// TIA Portal project "PrensaPiezas" (V18)

(* hardware
DEVICE "S7-1200 station_1"  S7-1200 Station
   slot 0: "Rack_0"  S7-1200 Rack  Rack  V1.0
   slot 1: "PLC_1"  CPU 1214C AC/DC/Rly  6ES7 214-1BG40-0XB0  V4.6
*)

// ===== PLC "PLC_1"  CPU 1214C AC/DC/Rly =====

VAR_GLOBAL   // PLC tag table "Default tag table"
   "rampa" AT %I0.0 : Bool;   // Sensor del objeto al caer de la rampa
   "zonaPrensa" AT %I0.1 : Bool;   // Sensor de la zona de la prensa
   "piezaPosicion" AT %I0.2 : Bool;   // Sensor de la pieza en posicion
   "prensa" AT %I0.3 : Bool;   // Sensor de la prensa
   "finalTramo" AT %I0.4 : Bool;   // Sensor del tramo final de la cinta
   "cintaAvanza" AT %M0.0 : Bool;   // Marca para avanzar la cinta
   "centraPieza" AT %M0.1 : Bool;   // Marca para centrar la pieza
   "cilindroBaja" AT %M0.2 : Bool;   // Marca para accionar la prensa
   "cintaRetrocede" AT %M0.3 : Bool;   // Marca para retroceder la cinta
   "guiaFlanco" AT %M0.4 : Bool;   // Marca guia de flanco
   "guiaFlanco_1" AT %M0.5 : Bool;   // Marca guia de flanco
   "guiaFlanco_2" AT %M0.6 : Bool;   // Marca guia de flanco
   "guiaFlanco_3" AT %M0.7 : Bool;   // Marca guia de flanco
   "motor" AT %Q0.0 : Bool;   // Motor hacia delante
   "motor_2" AT %Q0.1 : Bool;   // Motor hacia atras
   "presadoPieza" AT %Q0.2 : Bool;   // Prensado a la pieza
   "centrarPieza" AT %Q0.3 : Bool;   // Centrador de la pieza
END_VAR

// folder: System blocks/Program resources

DATA_BLOCK "retardoPiezaPresado"   // DB1
{ S7_Optimized_Access := 'TRUE' }
AUTHOR : Simatic
FAMILY : IEC
NAME : IEC_TMR
VERSION : 1.0
// stored: InstanceOfName IEC_TIMER
"IEC_TIMER"
BEGIN
END_DATA_BLOCK

// folder: (top level)

ORGANIZATION_BLOCK "Main"   // OB1, LAD, ProgramCycle
TITLE = "Main Program Sweep (Cycle)"
{ S7_Optimized_Access := 'TRUE' }
VERSION : 0.1
   VAR_INPUT
      Initial_Call : Bool;   // Initial call of this OB
      Remanence : Bool;   // =True, if remanent data are available
   END_VAR
   VAR_TEMP   // added for the SCL form of the ladder/FBD networks
      _w1 : Bool;
      _w2 : Bool;
   END_VAR
BEGIN

REGION Network 1: Marca para avanzar la cinta
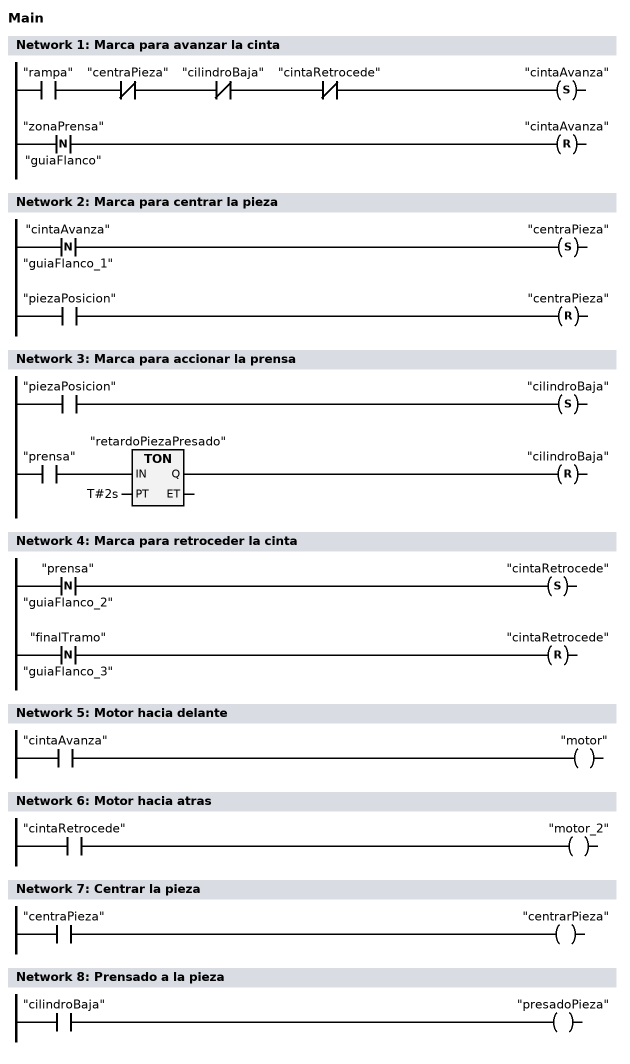
   RUNG wire#powerrail
      Contact( "rampa" )
      I_Contact( "centraPieza" )
      I_Contact( "cilindroBaja" )
      I_Contact( "cintaRetrocede" )
      S_Coil( "cintaAvanza" )
   END_RUNG
   RUNG wire#powerrail
      N_Contact(operand := "zonaPrensa", bit := "guiaFlanco")
      R_Coil( "cintaAvanza" )
   END_RUNG
   // the same network as SCL:
   IF "rampa" AND NOT "centraPieza" AND NOT "cilindroBaja" AND NOT "cintaRetrocede" THEN
       "cintaAvanza" := TRUE;
   END_IF;
   #_w1 := NOT "zonaPrensa" AND "guiaFlanco";   // falling edge of "zonaPrensa"
   "guiaFlanco" := "zonaPrensa";
   IF #_w1 THEN "cintaAvanza" := FALSE; END_IF;
END_REGION

REGION Network 2: Marca para centrar la pieza
   RUNG wire#powerrail
      N_Contact(operand := "cintaAvanza", bit := "guiaFlanco_1")
      S_Coil( "centraPieza" )
   END_RUNG
   RUNG wire#powerrail
      Contact( "piezaPosicion" )
      R_Coil( "centraPieza" )
   END_RUNG
   // the same network as SCL:
   #_w1 := NOT "cintaAvanza" AND "guiaFlanco_1";   // falling edge of "cintaAvanza"
   "guiaFlanco_1" := "cintaAvanza";
   IF #_w1 THEN "centraPieza" := TRUE; END_IF;
   IF "piezaPosicion" THEN "centraPieza" := FALSE; END_IF;
END_REGION

REGION Network 3: Marca para accionar la prensa
   IF "piezaPosicion" THEN "cilindroBaja" := TRUE; END_IF;
   "retardoPiezaPresado".TON(IN := "prensa", PT := T#2s);
   IF "retardoPiezaPresado".Q THEN "cilindroBaja" := FALSE; END_IF;
END_REGION

REGION Network 4: Marca para retroceder la cinta
   RUNG wire#powerrail
      N_Contact(operand := "prensa", bit := "guiaFlanco_2")
      S_Coil( "cintaRetrocede" )
   END_RUNG
   RUNG wire#powerrail
      N_Contact(operand := "finalTramo", bit := "guiaFlanco_3")
      R_Coil( "cintaRetrocede" )
   END_RUNG
   // the same network as SCL:
   #_w1 := NOT "prensa" AND "guiaFlanco_2";   // falling edge of "prensa"
   "guiaFlanco_2" := "prensa";
   IF #_w1 THEN "cintaRetrocede" := TRUE; END_IF;
   #_w2 := NOT "finalTramo" AND "guiaFlanco_3";   // falling edge of "finalTramo"
   "guiaFlanco_3" := "finalTramo";
   IF #_w2 THEN "cintaRetrocede" := FALSE; END_IF;
END_REGION

REGION Network 5: Motor hacia delante
   RUNG wire#powerrail
      Contact( "cintaAvanza" )
      Coil( "motor" )
   END_RUNG
   // the same network as SCL:
   "motor" := "cintaAvanza";
END_REGION

REGION Network 6: Motor hacia atras
   RUNG wire#powerrail
      Contact( "cintaRetrocede" )
      Coil( "motor_2" )
   END_RUNG
   // the same network as SCL:
   "motor_2" := "cintaRetrocede";
END_REGION

REGION Network 7: Centrar la pieza
   RUNG wire#powerrail
      Contact( "centraPieza" )
      Coil( "centrarPieza" )
   END_RUNG
   // the same network as SCL:
   "centrarPieza" := "centraPieza";
END_REGION

REGION Network 8: Prensado a la pieza
   RUNG wire#powerrail
      Contact( "cilindroBaja" )
      Coil( "presadoPieza" )
   END_RUNG
   // the same network as SCL:
   "presadoPieza" := "cilindroBaja";
END_REGION
END_ORGANIZATION_BLOCK